           IF (NOT #xDriveEnable_IC) OR #xDriveError THEN
               // Merker für Positionieren zurücksetzen
               #xProfileStart_IC := FALSE;
               #xProfileRestart_IC := FALSE;
               #xProfileStart_IC := FALSE;
               #xProfileActive := FALSE;
               #xHomingStart_IC := False;
               #xHomingSet_IC := FALSE;
               #xManualPos_IC := FALSE;
               #xManualPos_IC := FALSE;
               // wProfileNumberSet_IC := 1;    entfallen mit V1.1        
           END_IF;




           // Steuerdaten zuweisen
           #scInternalCtrl94.b0 := NOT #xDriveEnable_IC;
           #scInternalCtrl94.b1 := #xDriveSetQsp_IC;
           #scInternalCtrl94.b2 := #xEnablePositionTeach_IC;
           #scInternalCtrl94.b3 := #xHomingStart_IC;
           #scInternalCtrl94.b4 := #xHomingReset_IC;
           #scInternalCtrl94.b5 := #xProfileActive OR #xProfileStart_IC;
           #scInternalCtrl94.b6 := #xProfileStart_IC AND NOT #xProfilePosStop_IC;
           #scInternalCtrl94.b7 := #xProfileRestart_IC AND NOT #xProfilePosStop_IC;
           #scInternalCtrl94.b8 := #xProfileReset_IC;
           #scInternalCtrl94.b9 := #xEnableSpeedOverride_IC;
           #scInternalCtrl94.b10 := #xResetError_IC;
           #scInternalCtrl94.b11 := False; // Spare Set Error
           #scInternalCtrl94.b12 := #xHomingSet_IC;
           #scInternalCtrl94.b13 := False; // Spare
           #scInternalCtrl94.b14 := #xManualPos_IC;
           #scInternalCtrl94.b15 := #xManualNeg_IC;

           // zuweisen der freien Controlbits
           #wOUT := 0;  // Initialisierung
           #xwOut[8] := #xFreeCtrl_1_IC;
           #xwOut[9] := #xFreeCtrl_2_IC;
           #xwOut[10] := #xFreeCtrl_3_IC;
           #xwOut[11] := #xFreeCtrl_4_IC;
           #xwOut[12] := #xFreeCtrl_5_IC;
           #xwOut[13] := #xFreeCtrl_6_IC;
           #xwOut[14] := #xFreeCtrl_7_IC;
           #xwOut[15] := #xFreeCtrl_8_IC;
           #scInternalCtrl94.awInt[6] := #wOUT;
           #scInternalCtrl94.awInt[7] := #wFreeCtrl_1_IC;



           // limit rSpeedOverride
           #rSpeedOverrideSet_IC := LIMIT(MN := 0.0, IN := #rSpeedOverrideSet_IC, MX := 199.0);
           // scale and Write rSpeedOverride to drive
           IF #xEnableSpeedOverride_IC THEN
               #scInternalCtrl94.awInt[2] := INT_TO_WORD(REAL_TO_INT(#rSpeedOverrideSet_IC * 163.84));
           ELSE
               #scInternalCtrl94.awInt[2] := 16384;
           END_IF;
           // convert units to increments    
         //ABS :-)  #dwTemp := #AxisData.%DBD68; // DB SetAxisData.rUnitsToPos
         //ABS :-)  #rTemp := DWORD_TO_REAL(#dwTemp);
           #diSetPos := REAL_TO_DINT(#rPositionSet_IC * #i_stcAxisData.rUnitsToPos );//#rTemp);

           // write to drive*)
           #scInternalCtrl94.awInt[4] := DINT_TO_WORD(#diSetPos);
           #scInternalCtrl94.awInt[3] := DWORD_TO_WORD(SHR(IN := DINT_TO_DWORD(#diSetPos), N := 16));

           // limit  ProfileNumber and write To Drive      
           #scInternalCtrl94.awInt[5] := INT_TO_WORD(LIMIT(MN := 1, IN := WORD_TO_INT(#wProfileNumberSet_IC), MX := 75));

           // Ausgangsdaten zum Regler schreiben                         
           #iWriteError := DPWR_DAT(
                                    LADDR := #tHW_IO,
                                    RECORD := #scInternalCtrl94);

           #xError := (#iReadError <> 0) OR (#iWriteError <> 0)
           OR NOT ((#iDriveType <> 1) OR (#iDriveType <> 2) OR (#iDriveType <> 11))
           OR (WORD_TO_INT(#wProfileNumberSet_IC) > 75)
           OR (WORD_TO_INT(#wProfileNumberSet_IC) < 1);


       ELSE:
           #xError := True;
   END_CASE;






   IF (#iReadError <> 0) OR (#iWriteError <> 0) THEN
       #xCommunicationOK:=false;
   ELSE
       #xCommunicationOK:=True;
   END_IF;
END_FUNCTION_BLOCK

FUNCTION_BLOCK "LCB_12x_SetAxisData"   // FB443, SCL
{ S7_Optimized_Access := 'FALSE' }
AUTHOR : Lenze
FAMILY : LCB
NAME : SetAxisD
VERSION : 1.0
   VAR_INPUT
      rFeedConstant : Real := 3.6e+2;
      rCycleLength : Real := 3.6e+2;
      diGearNumerator : DInt := L#1;
      diGearDenominator : DInt := L#1;
      rReferenceSpeed : Real := 1.8e+5;
      rReferenceTorque : Real := 1.0e+0;
      sAxisName : String[16] := 'MyAxis';
      rResolution : Real := 16.0;
   END_VAR
   VAR_OUTPUT
      AxisData : "stcLCB_12x_SetAxisData_Sw";
   END_VAR
   VAR_IN_OUT
      xModeUnlimited : Bool := TRUE;
      xModeLimited : Bool;
      xModeModulo : Bool;
   END_VAR
   VAR
      rInvFeedConstant : Real;
      diReferenceSpeed_s : DInt;
      rEncoderGear : Real;
      rInvEncoderGear : Real;
      diCycleLength_p : DInt;
      rUnitsToPos : Real;
      rPosToUnits : Real;
      rUnitsToSpeed : Real;
      rSpeedToUnits : Real;
      rTimeUnit : Real := 6.0e+1;
      rFeedConstantOld : Real;
      rCycleLengthOld : Real;
      diGearNumeratorOld : DInt := L#2;
      diGearDenominatorOld : DInt := L#2;
      rReferenceSpeedOld : Real;
      rResolutionOld : Real := 1.0;
      xModeUnlimitedOld : Bool;
      xModeLimitedOld : Bool;
      xModeModuloOld : Bool;
   END_VAR
BEGIN

       IF #xModeUnlimited= True THEN #xModeLimited:= False; #xModeModulo:= False;
           ELSIF #xModeLimited= True THEN #xModeUnlimited:= False; #xModeModulo:= False;
               ELSIF #xModeModulo= True THEN #xModeUnlimited:= False; #xModeLimited:= False;
       END_IF; 
       IF ((#rFeedConstantOld <> #rFeedConstant) OR
           (#diGearNumeratorOld <> #diGearNumerator) OR
           (#diGearDenominatorOld <> #diGearDenominator) OR
           (#rCycleLengthOld <> #rCycleLength) OR
           (#xModeUnlimitedOld <> #xModeUnlimited) OR
           (#xModeLimitedOld <> #xModeLimited) OR
           (#xModeModuloOld <> #xModeModulo) OR
           (#rResolutionOld <> #rResolution) OR
           (#rReferenceSpeedOld <> #rReferenceSpeed)) THEN


           #rInvFeedConstant := 1.0 / #rFeedConstant;

       (* Achsdatenberechnung starten *)
       (* Getriebefaktor *)
           #rEncoderGear:=DINT_TO_REAL(#diGearNumerator) / DINT_TO_REAL(#diGearDenominator);
           #rInvEncoderGear:= 1.0 / #rEncoderGear;
       (* Umrechenfaktor Units -> _p bestimmen *)
           #rUnitsToPos := (#rInvFeedConstant * #rEncoderGear) * (2**#rResolution);
       (* Umrechenfaktor _p -> Units bestimmen *)
           #rPosToUnits := 1.0 / #rUnitsToPos;
       (* Umrechenfaktor Units->_s bestimmen *)
           #rUnitsToSpeed := #rInvFeedConstant * #rEncoderGear;
     //  (* mal 2^32 (eine Umdrehung) *)
     //      rUnitsToSpeed := rUnitsToSpeed * 2**32;
       (* durch Zeiteinheit teilen *)
           #rUnitsToSpeed := #rUnitsToSpeed * #rTimeUnit;
       (* Umrechenfaktor _s -> Units bestimmen *)
           #rSpeedToUnits := 1.0 / #rUnitsToSpeed;
       (*Referenzgeschwindigkeit bestimmen *)
           #diReferenceSpeed_s := REAL_TO_DINT(#rReferenceSpeed * #rUnitsToSpeed);

           IF #xModeModulo THEN
               #diCycleLength_p := REAL_TO_DINT(#rCycleLength * #rUnitsToPos) ;
           ELSE
               #diCycleLength_p := 0;
           END_IF;

       // sichern der aktuellen Werte für Änderungsvergleich
           #rFeedConstantOld     :=#rFeedConstant     ;
           #rCycleLengthOld      :=#rCycleLength      ;    
           #diGearNumeratorOld   :=#diGearNumerator   ;
           #diGearDenominatorOld :=#diGearDenominator ;
           #rReferenceSpeedOld   :=#rReferenceSpeed   ;
           #xModeUnlimitedOld    :=#xModeUnlimited    ;
           #xModeLimitedOld      :=#xModeLimited      ;
           #xModeModuloOld       :=#xModeModulo       ;
           #rResolutionOld      :=#rResolution      ;  

       END_IF;

   //Write to global output status
       #AxisData.rUnitsToPos := #rUnitsToPos;
       #AxisData.rPosToUnits := #rPosToUnits;
END_FUNCTION_BLOCK